TYPE ST_SoftSettings :
STRUCT
	{ attribute 'TcHmiSymbol.ShowRecursively' }
	inputgrid					: ST_SoftSettings_Grid;
	inputgenset					: ST_SoftSettings_Genset;
	PSB							: ST_SoftSettings_Peakshavebox;
	ACDCcharger					: ST_Softsettings_ACDCcharger;
	{ attribute 'TcHmiSymbol.ShowRecursively' }
	system						: ST_SoftSettings_System;
	setup						: ST_SoftSettings_Setup;
END_STRUCT
END_TYPE

(* stored: Version 1.1.0.1, ProductVersion 3.1.4024.12
   DUT ST_SoftSettings: Id {aa1c06b3-e538-4ac2-ad62-86bb97d9209a} *)
